// TIA Portal V20 export
VAR_GLOBAL   // PLC tag table "Default tag table"
   All_Lamps AT %QB0 : Byte;
   Lamps_On AT %Q5.0 : Bool;
   Light2State AT %M0.0 : Bool;
   Light1State AT %M0.1 : Bool;
   Light3State AT %M0.2 : Bool;
   LightStep AT %MW0 : Int;
   start AT %M2.0 : Bool;
   Elapsed_Time AT %MD4 : Time;
   Lamps AT %MB0 : Byte;
END_VAR
